FUNCTION_BLOCK fb_lensTranport
VAR_INPUT
END_VAR
VAR_OUTPUT
END_VAR
VAR
	SFCInit: bool;
	trn_wattingForLensDone: BOOL;
	trn_connectionCheckDone: BOOL;
	flg_buf_gateLengthISSuccessed: BOOL;
	flg_buf_dummySignal: BOOL;
	trn_chuckDone: BOOL;
	var_chuckCount: INT;
	trn_transportDone: BOOL;
	trn_waitTakingLensDone: BOOL;
	trn_moveToHomeDone: BOOL;
	fbi_getCav: fb_getCav;
	trn_readCavDone: BOOL;
	trn_gm_chuckDone: BOOL;
	trn_gm_transportDone: BOOL;
	trn_gm_moveToHomeDone: BOOL;
	trn_cavCheckDone: BOOL;
	fbi_delayTimer: TON;
	trn_AddCountDone: BOOL;
	var_process: INT;
	flg_chuckDone: BOOL;
	flg_pushDone: BOOL;
	trn_LensCheckDone: BOOL;
END_VAR

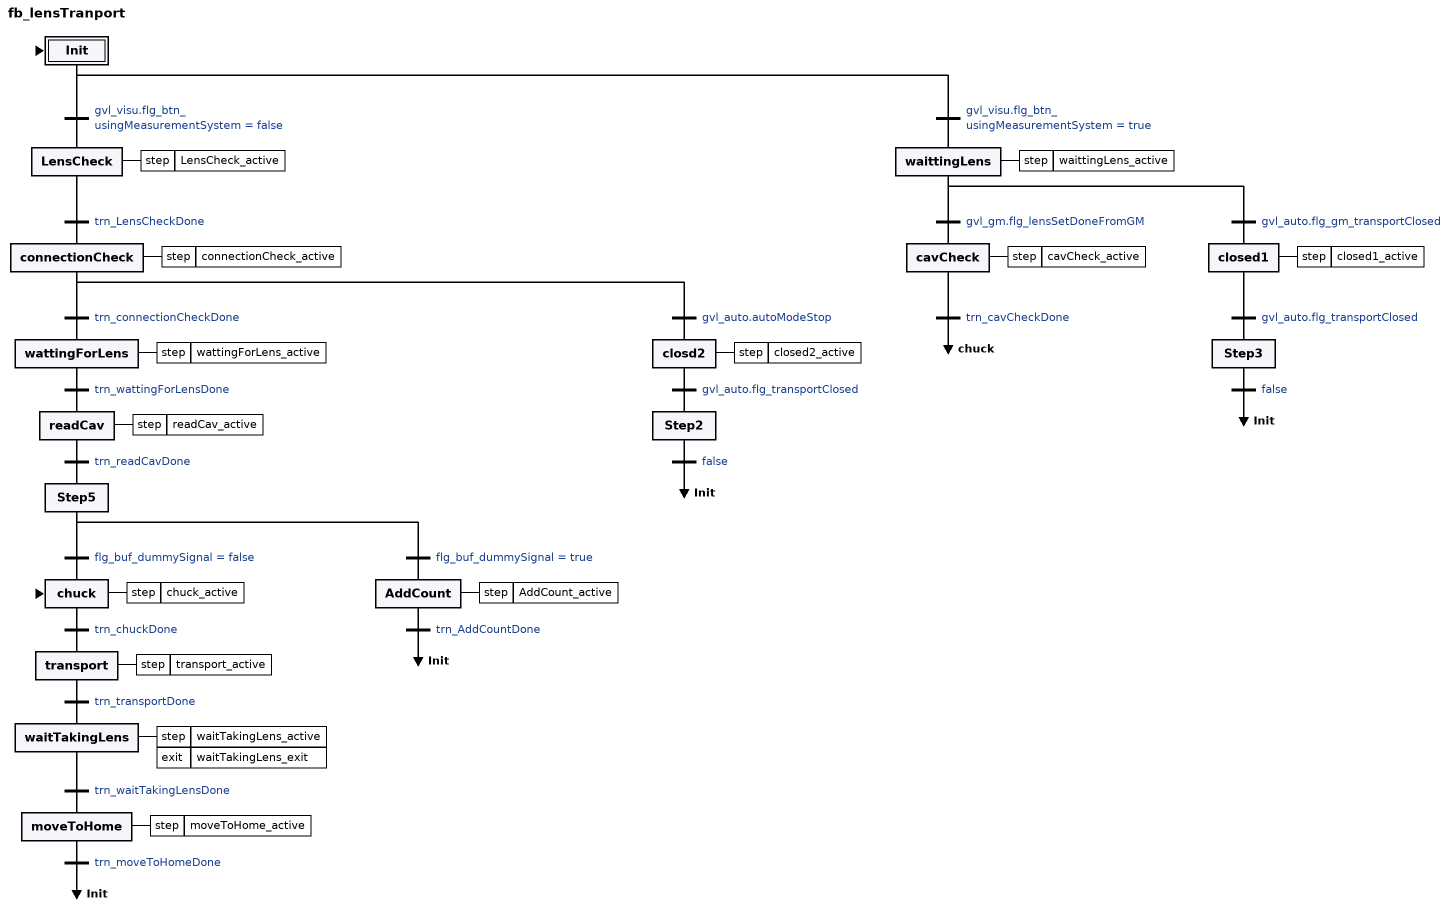
INITIAL_STEP Init:
END_STEP
TRANSITION FROM Init TO LensCheck
    := gvl_visu.flg_btn_usingMeasurementSystem = false;
END_TRANSITION
TRANSITION FROM Init TO waittingLens
    := gvl_visu.flg_btn_usingMeasurementSystem = true;
END_TRANSITION
STEP waittingLens:
    waittingLens_active(N);  // step action
END_STEP
TRANSITION FROM waittingLens TO cavCheck
    := gvl_gm.flg_lensSetDoneFromGM;
END_TRANSITION
STEP cavCheck:
    cavCheck_active(N);  // step action
END_STEP
TRANSITION FROM cavCheck TO chuck
    := trn_cavCheckDone;
END_TRANSITION
TRANSITION FROM waittingLens TO closed1
    := gvl_auto.flg_gm_transportClosed;
END_TRANSITION
STEP closed1:
    closed1_active(N);  // step action
END_STEP
TRANSITION FROM closed1 TO Step3
    := gvl_auto.flg_transportClosed;
END_TRANSITION
STEP Step3:
END_STEP
TRANSITION FROM Step3 TO Init
    := false;
END_TRANSITION
STEP LensCheck:
    LensCheck_active(N);  // step action
END_STEP
TRANSITION FROM LensCheck TO connectionCheck
    := trn_LensCheckDone;
END_TRANSITION
STEP connectionCheck:
    connectionCheck_active(N);  // step action
END_STEP
TRANSITION FROM connectionCheck TO wattingForLens
    := trn_connectionCheckDone;
END_TRANSITION
STEP wattingForLens:
    wattingForLens_active(N);  // step action
END_STEP
TRANSITION FROM wattingForLens TO readCav
    := trn_wattingForLensDone;
END_TRANSITION
TRANSITION FROM connectionCheck TO closd2
    := gvl_auto.autoModeStop;
END_TRANSITION
STEP closd2:
    closed2_active(N);  // step action
END_STEP
TRANSITION FROM closd2 TO Step2
    := gvl_auto.flg_transportClosed;
END_TRANSITION
STEP Step2:
END_STEP
TRANSITION FROM Step2 TO Init
    := false;
END_TRANSITION
STEP readCav:
    readCav_active(N);  // step action
END_STEP
TRANSITION FROM readCav TO Step5
    := trn_readCavDone;
END_TRANSITION
STEP Step5:
END_STEP
TRANSITION FROM Step5 TO chuck
    := flg_buf_dummySignal = false;
END_TRANSITION
TRANSITION FROM Step5 TO AddCount
    := flg_buf_dummySignal = true;
END_TRANSITION
STEP AddCount:
    AddCount_active(N);  // step action
END_STEP
TRANSITION FROM AddCount TO Init
    := trn_AddCountDone;
END_TRANSITION
STEP chuck:
    chuck_active(N);  // step action
END_STEP
TRANSITION FROM chuck TO transport
    := trn_chuckDone;
END_TRANSITION
STEP transport:
    transport_active(N);  // step action
END_STEP
TRANSITION FROM transport TO waitTakingLens
    := trn_transportDone;
END_TRANSITION
STEP waitTakingLens:
    waitTakingLens_active(N);  // step action
    waitTakingLens_exit(P0);  // exit action
END_STEP
TRANSITION FROM waitTakingLens TO moveToHome
    := trn_waitTakingLensDone;
END_TRANSITION
STEP moveToHome:
    moveToHome_active(N);  // step action
END_STEP
TRANSITION FROM moveToHome TO Init
    := trn_moveToHomeDone;
END_TRANSITION

ACTION AddCount_active:
IF AddCount._x AND AddCount.x = FALSE THEN
	trn_AddCountDone := FALSE;
ELSIF AddCount._x AND AddCount.x THEN
	trn_AddCountDone := TRUE;
END_IF
END_ACTION

ACTION cavCheck_active:
IF cavCheck._x AND cavCheck.x = FALSE THEN
	trn_cavCheckDone := FALSE;
ELSIF cavCheck._x AND cavCheck.x THEN
	gvl_auto.cavNo := gvl_gm.var_buf_tranportCav;
	gvl_auto.flg_buf_gateLengthIsPassed := gvl_gm.flg_buf_gateLengthIsPassed;
	trn_cavCheckDone := TRUE;
END_IF
END_ACTION

ACTION chuck_active:
IF chuck._x AND chuck.x = FALSE THEN
	gvl_gm.flg_lensRequest := FALSE;
	trn_chuckDone := FALSE;
	gvl_auto.flg_gateData_Tx := FALSE;
	gvl_solv.fbi_chuck.in_flg_run := FALSE;
	gvl_solv.fbi_push.in_flg_run := FALSE;
	var_chuckCount := -11;
ELSIF chuck._x AND chuck.x THEN
	CASE var_chuckCount OF
		-11:
			IF gvl_param.var_productInfo[gvl_param.var_currentProductID].flg_mode_stocker THEN
				var_chuckCount := -10; // Mode 1
			ELSE
				var_chuckCount := 0;  // Mode 0
			END_IF
		
		// Mode 1: 押す →　解除　→ チャック →　押す
		-10:
			gvl_solv.fbi_push.in_var_moveMode := eP_svMoveMode.svB;
			gvl_solv.fbi_push.in_flg_run := TRUE;
			var_chuckCount := -9;
		-9://close
			IF gvl_solv.fbi_push.out_flg_Done THEN
				gvl_solv.fbi_push.in_flg_run := FALSE;
				var_chuckCount := -8;
			END_IF
		-8:		
			gvl_solv.fbi_push.in_var_moveMode := eP_svMoveMode.svA;
			gvl_solv.fbi_push.in_flg_run := TRUE;
			var_chuckCount := -7;
		-7://open
			IF gvl_solv.fbi_push.out_flg_Done THEN
				gvl_solv.fbi_push.in_flg_run := FALSE;
				var_chuckCount := -6;
			END_IF
		-6:
			gvl_solv.fbi_chuck.in_var_moveMode := eP_svMoveMode.svB;
			gvl_solv.fbi_chuck.in_flg_run := TRUE;
			var_chuckCount := -5;
		-5://push close
			IF gvl_solv.fbi_chuck.out_flg_Done THEN
				gvl_solv.fbi_chuck.in_flg_run := FALSE;
				var_chuckCount := -4;
			END_IF
		-4:
			gvl_solv.fbi_push.in_var_moveMode := eP_svMoveMode.svB;
			gvl_solv.fbi_push.in_flg_run := TRUE;
			var_chuckCount := -3;
		-3://close
			
			IF gvl_solv.fbi_push.out_flg_Done THEN
				gvl_solv.fbi_push.in_flg_run := FALSE;
				var_chuckCount := 12;
			END_IF
		
		// Mode 0: チャック → 解除 → 押す → チャック
		0:
			gvl_solv.fbi_chuck.in_var_moveMode := eP_svMoveMode.svB;
			gvl_solv.fbi_chuck.in_flg_run := TRUE;
			var_chuckCount := 1;
		1://close
			
			IF gvl_solv.fbi_chuck.out_flg_Done THEN
				gvl_solv.fbi_chuck.in_flg_run := FALSE;
				var_chuckCount := 2;
			END_IF
		2:		
			gvl_solv.fbi_chuck.in_var_moveMode := eP_svMoveMode.svA;
			gvl_solv.fbi_chuck.in_flg_run := TRUE;
			var_chuckCount := 3;
		3://open
			
			IF gvl_solv.fbi_chuck.out_flg_Done THEN
				var_chuckCount := 4;
			END_IF
		4:
			gvl_solv.fbi_push.in_var_moveMode := eP_svMoveMode.svB;
			gvl_solv.fbi_push.in_flg_run := TRUE;
			var_chuckCount := 5;
		5://push close
			
			IF gvl_solv.fbi_push.out_flg_Done THEN
				gvl_solv.fbi_push.in_flg_run := FALSE;
				gvl_solv.fbi_chuck.in_flg_run := FALSE;
				var_chuckCount := 6;
			END_IF
		6:
			
			gvl_solv.fbi_chuck.in_var_moveMode := eP_svMoveMode.svB;
			gvl_solv.fbi_chuck.in_flg_run := TRUE;
			var_chuckCount := 7;
		7://close
			
			IF gvl_solv.fbi_chuck.out_flg_Done THEN
				gvl_solv.fbi_chuck.in_flg_run := FALSE;
				var_chuckCount := 12;
			END_IF
		8:
			
			gvl_solv.fbi_chuck.in_var_moveMode := eP_svMoveMode.svA;
			gvl_solv.fbi_chuck.in_flg_run := TRUE;
			var_chuckCount := 9;
		9://open
			
			IF gvl_solv.fbi_chuck.out_flg_Done THEN
				gvl_solv.fbi_chuck.in_flg_run := FALSE;
				var_chuckCount := 10;
			END_IF
		10:
			
			gvl_solv.fbi_chuck.in_var_moveMode := eP_svMoveMode.svB;
			gvl_solv.fbi_chuck.in_flg_run := TRUE;
			var_chuckCount := 11;
		11://close
			
			IF gvl_solv.fbi_chuck.out_flg_Done THEN
				var_chuckCount := 12;
			END_IF
		12://gate measurement
			IF gvl_visu.flg_btn_gateMeasurementIsNone THEN
				IF flg_buf_gateLengthISSuccessed THEN
					gvl_auto.gateLengthIsPassed := TRUE;
				ELSIF gvl_auto.flg_buf_gateLengthIsPassed THEN
					gvl_auto.gateLengthIsPassed := TRUE;
				ELSE
					gvl_auto.gateLengthIsPassed := FALSE;
				END_IF
			ELSE
				IF gvl_io.var_gateLength > gvl_param.var_productInfo[gvl_param.var_currentProductID].gateLength_max OR gvl_io.var_gateLength < gvl_param.var_productInfo[gvl_param.var_currentProductID].gateLength_min THEN
					gvl_auto.gateLengthIsPassed := FALSE;
				ELSE
					gvl_auto.gateLengthIsPassed := TRUE;
				END_IF
				gvl_auto.flg_gateData_Tx := TRUE;
				
			END_IF
			var_chuckCount := 13;
		13:
			gvl_solv.fbi_chuck.in_flg_run := FALSE;
			gvl_elecylinder.fbi_axisRotary.in_flg_run := FALSE;
			gvl_elecylinder.fbi_axisRotary.in_var_moveMode := eP_eleMoveMode.eleB;
			IF gvl_visu.flg_btn_RotaryIsNotUse THEN
				var_chuckCount := 16;
			ELSE
				var_chuckCount := 14;
			END_IF
		14:
			gvl_elecylinder.fbi_axisRotary.in_flg_run := TRUE;
			var_chuckCount := 15;
		15:
			IF gvl_elecylinder.fbi_axisRotary.out_flg_Done THEN
				gvl_elecylinder.fbi_axisRotary.in_flg_run := FALSE;
				var_chuckCount := 16;
			END_IF
		16:
			trn_chuckDone := TRUE;
	END_CASE
END_IF
END_ACTION

ACTION closed1_active:
IF closed1._x AND closed1.x = FALSE THEN
	gvl_auto.flg_transportClosed := FALSE;
	gvl_elecylinder.fbi_axisTransport.in_flg_run := FALSE;
	gvl_elecylinder.fbi_axisRotary.in_flg_run:= FALSE;
	gvl_elecylinder.fbi_axisTransport.in_var_moveMode := eP_eleMoveMode.eleB;
	gvl_elecylinder.fbi_axisRotary.in_var_moveMode:= eP_eleMoveMode.eleB;
	var_process := 0;
ELSIF closed1._x AND closed1.x THEN
	CASE var_process OF
		0:
			gvl_elecylinder.fbi_axisRotary.in_flg_run:= TRUE;
			var_process := 1;
		1:
			IF gvl_elecylinder.fbi_axisRotary.out_flg_Done THEN
				gvl_elecylinder.fbi_axisRotary.in_flg_run:= FALSE;
				var_process := 2;
			END_IF
		2:
			gvl_elecylinder.fbi_axisTransport.in_flg_run := TRUE;
			var_process := 3;
		3:
			IF gvl_elecylinder.fbi_axisTransport.out_flg_Done THEN
				gvl_elecylinder.fbi_axisTransport.in_flg_run:= FALSE;
				gvl_auto.flg_transportClosed := TRUE;
			END_IF
	END_CASE
END_IF
END_ACTION

ACTION closed2_active:
IF closd2._x AND closd2.x = FALSE THEN
	gvl_auto.flg_transportClosed := FALSE;
ELSIF closd2._x AND closd2.x THEN
	gvl_io.flg_requestLens := FALSE;
	gvl_auto.flg_transportClosed := true;
END_IF
END_ACTION

ACTION connectionCheck_active:
IF connectionCheck._x AND connectionCheck.x = FALSE THEN
	trn_connectionCheckDone:= FALSE;
	gvl_io.flg_requestLens := TRUE;
ELSIF connectionCheck._x AND connectionCheck.x THEN
	IF gvl_io.in_bitNumber0 
		AND gvl_io.in_bitNumber1
		AND gvl_io.in_bitNumber2
		AND gvl_io.in_bitNumber3 OR gvl_debug.cavConecctSkip THEN
		trn_connectionCheckDone:= TRUE;
	END_IF
	IF NOT gvl_visu.flg_btn_vacSensOn THEN
		gvl_error.flg_fiberSens := gvl_io.flg_fiberSens;
	END_IF
END_IF
END_ACTION

ACTION LensCheck_active:
IF LensCheck._x AND LensCheck.x = FALSE THEN
	trn_LensCheckDone := FALSE;
ELSIF LensCheck._x AND LensCheck.x THEN
	IF NOT gvl_visu.flg_btn_vacSensOn THEN
		IF gvl_io.flg_fiberSens OR gvl_debug.out_fiberSens THEN
			gvl_error.flg_fiberSens := TRUE;	
		ELSE
			trn_LensCheckDone := TRUE;
		END_IF
	ELSE
		trn_LensCheckDone := TRUE;
	END_IF
END_IF
END_ACTION

ACTION moveToHome_active:
IF moveToHome._x AND moveToHome.x = FALSE THEN
	trn_moveToHomeDone := FALSE;
	gvl_elecylinder.fbi_axisTransport.in_flg_run := FALSE;
	gvl_elecylinder.fbi_axisTransport.in_var_moveMode := eP_eleMoveMode.eleA;
	gvl_elecylinder.fbi_axisRotary.in_var_moveMode := eP_eleMoveMode.eleA;
	var_process := 0;
ELSIF moveToHome._x AND moveToHome.x THEN
	CASE var_process OF
		0:
			gvl_elecylinder.fbi_axisTransport.in_flg_run := TRUE;
			var_process := 1;
		1:
			IF gvl_elecylinder.fbi_axisTransport.out_flg_Done THEN
				gvl_elecylinder.fbi_axisTransport.in_flg_run := FALSE;
				var_process := 2;
			END_IF
		2:
			gvl_elecylinder.fbi_axisRotary.in_flg_run := TRUE;
			var_process := 3;
		3:
			IF gvl_elecylinder.fbi_axisRotary.out_flg_Done THEN
				gvl_elecylinder.fbi_axisRotary.in_flg_run := FALSE;
				var_process := 4;
			END_IF
		4:
			IF gvl_elecylinder.ref_axis_transport.input.in_flg_sensA AND gvl_elecylinder.ref_axis_rotary.input.in_flg_sensA THEN
				trn_moveToHomeDone := TRUE;
			END_IF
	END_CASE
	
	
	//
END_IF
END_ACTION

PROPERTY p_Init : bool
GET
p_init := THIS^.SFCInit;
END_GET
SET
THIS^.SFCInit := p_init;
END_SET
END_PROPERTY

ACTION readCav_active:
IF readCav._x AND readCav.x = FALSE THEN
	trn_readCavDone := FALSE;
	THIS^.fbi_getCav();
	fbi_getCav.in_flg_run := FALSE;
	fbi_delayTimer.IN := FALSE;
ELSIF readCav._x AND readCav.x THEN
	THIS^.fbi_getCav();
	fbi_delayTimer.IN := TRUE;
	THIS^.fbi_getCav.in_flg_run := fbi_delayTimer.Q;
	IF THIS^.fbi_getCav.out_flg_Done THEN
		IF gvl_debug.flg_debug_run THEN
			gvl_auto.cavNo := gvl_debug.var_cav;
		ELSE
			gvl_auto.cavNo := THIS^.fbi_getCav.out_var_cav;
		END_IF
		trn_readCavDone := TRUE;
	ELSIF THIS^.fbi_getCav.out_flg_error THEN
		IF gvl_debug.flg_debug_run THEN
			gvl_auto.cavNo := gvl_debug.var_cav;
		ELSE
			gvl_auto.cavNo := 0;
		END_IF
		trn_readCavDone := TRUE;
	END_IF
END_IF

fbi_delayTimer(IN:= , PT:=T#200MS , Q=> , ET=> );
END_ACTION

ACTION transport_active:
IF transport._x AND transport.x = FALSE THEN
	gvl_elecylinder.fbi_axisTransport.in_flg_run := FALSE;
	trn_transportDone := FALSE;
	gvl_elecylinder.fbi_axisTransport.in_var_moveMode := eP_eleMoveMode.eleB;
	var_process := 0;
ELSIF transport._x AND transport.x THEN
	CASE var_process OF
		0:
			IF NOT gvl_auto.flg_sampling THEN
				gvl_elecylinder.fbi_axisTransport.in_flg_run := TRUE;
				var_process := 1;
			END_IF
		1:
			IF gvl_elecylinder.fbi_axisTransport.out_flg_Done THEN
				gvl_elecylinder.fbi_axisTransport.in_flg_run := FALSE;
				trn_transportDone := TRUE;
			END_IF
	END_CASE
END_IF
END_ACTION

ACTION waitTakingLens_active:
IF waitTakingLens._x AND waitTakingLens.x = FALSE THEN
	trn_waitTakingLensDone := FALSE;
	flg_chuckDone:= FALSE;
	flg_pushDone := FALSE;
	gvl_solv.fbi_chuck.in_var_moveMode := eP_svMoveMode.svA;
	gvl_solv.fbi_push.in_var_moveMode := eP_svMoveMode.svA;
	gvl_auto.buf_cavNo := gvl_auto.cavNo;
	gvl_auto.flg_gateLength := gvl_auto.gateLengthIsPassed;
ELSIF waitTakingLens._x AND waitTakingLens.x THEN
	gvl_auto.requirementToPickUpLens := TRUE;
	IF gvl_auto.lensVacuumDone THEN
		gvl_auto.buf_gateLength := gvl_visu.var_gateLengthList[0];
		gvl_solv.fbi_chuck.in_flg_run := TRUE;
		gvl_solv.fbi_push.in_flg_run := TRUE;
	END_IF
	IF gvl_solv.fbi_chuck.out_flg_Done THEN
		flg_chuckDone := TRUE;
	END_IF
	IF gvl_solv.fbi_push.out_flg_Done THEN
		flg_pushDone := TRUE;
	END_IF
	IF flg_chuckDone AND flg_pushDone THEN
		gvl_solv.fbi_chuck.in_flg_run := FALSE;
		gvl_solv.fbi_push.in_flg_run := FALSE;
		gvl_auto.chuckopenDone := TRUE;
	END_IF
	IF gvl_auto.pickUpLnesDone THEN
		trn_waitTakingLensDone := TRUE;
	END_IF
END_IF
END_ACTION

ACTION waitTakingLens_exit:
gvl_auto.lensVacuumDone := FALSE;
gvl_auto.requirementToPickUpLens := FALSE;
gvl_auto.chuckopenDone := FALSE;
gvl_auto.pickUpLnesDone := FALSE;
END_ACTION

ACTION waittingLens_active:
IF waittingLens._x AND waittingLens.x = FALSE THEN
	gvl_gm.flg_lensRequest := FALSE;
	gvl_gm.flg_lensSetDoneFromGM := FALSE;
	IF NOT gvl_visu.flg_btn_vacSensOn THEN
		gvl_error.flg_fiberSens := gvl_io.flg_fiberSens;
	END_IF
ELSIF waittingLens._x AND waittingLens.x THEN
	gvl_gm.flg_lensRequest := TRUE;
END_IF
END_ACTION

ACTION wattingForLens_active:
IF wattingForLens._x AND wattingForLens.x = FALSE THEN
	trn_wattingForLensDone := FALSE;
	flg_buf_gateLengthISSuccessed := FALSE;
	flg_buf_dummySignal := FALSE;
ELSIF wattingForLens._x AND wattingForLens.x THEN
	//gate
	IF gvl_IO.flg_gateLengthIsSuccessed OR gvl_debug.flg_passingMeasurement THEN
		flg_buf_gateLengthISSuccessed := TRUE;
	END_IF
	//dummy signal
	IF gvl_io.flg_dummySiganl THEN
		flg_buf_dummySignal := TRUE;
	END_IF
	//lens set done
	IF NOT gvl_visu.flg_btn_vacSensOn THEN
		IF gvl_io.flg_lensSetDone AND gvl_io.flg_fiberSens OR gvl_debug.out_lensSetDone THEN
			gvl_io.flg_requestLens := FALSE;
			trn_wattingForLensDone := TRUE;
		ELSIF gvl_io.flg_lensSetDone AND gvl_io.flg_fiberSens = FALSE THEN
			gvl_error.flg_fiberSens := TRUE;
		END_IF
	ELSE
		IF gvl_io.flg_lensSetDone OR gvl_debug.out_lensSetDone  THEN
			gvl_io.flg_requestLens := FALSE;
			trn_wattingForLensDone := TRUE;
		END_IF
	END_IF
END_IF
END_ACTION

END_FUNCTION_BLOCK

(* stored: Version 1.1.0.1, ProductVersion 3.1.4024.11
   POU fb_lensTranport: Id {1af97683-7a37-4f42-ad56-15d8586d31ec}, SpecialFunc None
   Action AddCount_active: Id {af952012-1912-4dcc-bdcc-6f9b4ca03ad5}
   Action cavCheck_active: Id {3bae6984-dd70-4894-81cb-6de1ca15a977}
   Action chuck_active: Id {143178f8-a408-4f7e-b700-2713719799ed}
   Action closed1_active: Id {3ff44ae3-cdf5-4730-b599-dc12571dc5e3}
   Action closed2_active: Id {de7f5a87-b624-45f6-a525-8a3d92b6d66a}
   Action connectionCheck_active: Id {86481e42-f6a3-457d-9c51-6beb53b6e46a}
   Action LensCheck_active: Id {750330bd-a01e-482d-ab83-669fd0e46480}
   Action moveToHome_active: Id {d2faca98-47cc-4672-a598-dab6972e62ac}
   Property p_Init: Id {27fa85b1-1531-4dcd-b935-6082f733efc7}
   Get Get: Id {ecc23f87-215f-49a9-af49-a92cd759bf69}
   Set Set: Id {ade26fc8-c356-45cf-89e6-dd1cb564c1cd}
   Action readCav_active: Id {b57bdeac-e9c8-464f-8c3b-b5f521852ea6}
   Action transport_active: Id {4f3b3e56-da30-4f7c-a4f4-e74a569115b0}
   Action waitTakingLens_active: Id {f1c88264-0288-4e61-bd47-dc6c375538ee}
   Action waitTakingLens_exit: Id {5ab854d4-b981-4cd4-b397-b9cb79adedb6}
   Action waittingLens_active: Id {96e5bade-22cb-40e2-be80-3360e92e96f1}
   Action wattingForLens_active: Id {1a897909-5b48-4c28-8a9a-28eadccb18cc} *)
